FUNCTION_BLOCK FB_TouchProbe_Home_Bylimit
VAR_INPUT	
		bCMD_HomeExecute			:REFERENCE TO BOOL;			(* 执行回零*)
		bCMD_Reset					:REFERENCE TO BOOL;			(* 回零错误复位*)
		bCMD_EnableState			:BOOL;						(* 使能状态输入*)	
		bCMD_StartHomeIndex			:BOOL;						(* 是否使用索引回零*)
		eCMD_HomeDirection			:MC_Direction;				(* 回原点方向*)
		bCMD_PositiveLimit			:BOOL;						(* 正限位传感器*)
		bCMD_NegativeLimit			:BOOL;						(* 负限位传感器*)
		rCMD_HomePosition			:LREAL;						(* 设定回原点位置*)
		rCMD_TowardsVelSetValue		:LREAL;						(* 靠近原点速度*)
		rCMD_OffVelSetValue			:LREAL;						(* 离开原点速度*)
	    stHomeAdsGroup				:ST_HomeAdsGroup;			(* ADS地址信息*)

END_VAR
VAR_OUTPUT
		bResult_HomeDone			:BOOL;						(* 回原点完成状态*)
		bResult_HomeBusy			:BOOL;						(* 正在回原点中状态*)
		bResult_HomeError			:BOOL;						(* 回原点错误状态*)
		nResult_HomeErrorID			:UDINT;						(* 回原点错误代码*)
END_VAR
VAR_IN_OUT
		axis						:AXIS_REF;
END_VAR
VAR
	  
		mcHome						:MC_Home;
		mcReset						:MC_Reset;
		fbReadParameter				:ARRAY [0..4] OF ADSREAD;
		fbwriteParameter			:ARRAY [0..4] OF ADSWRITE;
		rTowardsVelActValue			:LREAL;		
		rOffVelActValue				:LREAL;
		nHomeSenorSetValue			:INT;
		nHomeSensorActValue			:INT;
		nHomeSynSetValue			:WORD;
		nHomeSynActValue			:WORD;
		nHomeSetRefMode				:DINT;
		nHomeActRefMode				:DINT;
		mcHomeStatus				:ST_McOutputs;
		fbReadParaStatus			:ARRAY [0..4] OF ST_McOutputs;
		fbWriteParaStatus			:ARRAY [0..4] OF ST_McOutputs;
		posEdge_bCMD_HomeExecute	:R_TRIG;
		posEdge_bCMD_Reset			:R_TRIG;
		negEdge_bCMD_Calibration	:F_TRIG;
		ton_bCMD_HomeExecute		:TON;
		ton_nStep					:TON;
		ton_bCMD_Reset				:TON;
		ton_McReset					:TON;
		ton_HomErr                  :TON;
		nStep						:E_HomeStep;
		mcMoveAbs					:MC_MoveAbsolute;
END_VAR

posEdge_bCMD_HomeExecute(CLK:=bCMD_HomeExecute AND bCMD_EnableState AND NOT bResult_HomeError AND NOT bResult_HomeBusy);
ton_bCMD_HomeExecute(IN:=bCMD_HomeExecute,PT:=T#100MS);

IF posEdge_bCMD_HomeExecute.Q  THEN
	nStep:=AckHomeDirection;
ELSIF	ton_bCMD_HomeExecute.Q THEN
	 bCMD_HomeExecute:=FALSE;
END_IF


IF eCMD_HomeDirection=MC_Direction.MC_Positive_Direction  THEN
	mcHome.bCalibrationCam:=bCMD_PositiveLimit;
ELSIF eCMD_HomeDirection=MC_Direction.MC_Negative_Direction THEN
		mcHome.bCalibrationCam:=bCMD_NegativeLimit;
END_IF

CASE nStep OF
IndexHomeInital:
	ton_nStep(IN:=FALSE);		
	bResult_HomeBusy:=FALSE;
	mcHome.Execute:=FALSE;
	mcMoveAbs.Execute:=FALSE;
	fbReadParameter[0].READ:=fbReadParameter[1].READ:=fbReadParameter[2].READ:=fbReadParameter[3].READ:=fbReadParameter[4].READ:=FALSE;
	fbwriteParameter[0].WRITE:=fbwriteParameter[1].WRITE:=fbwriteParameter[2].WRITE:=fbwriteParameter[3].WRITE:=fbwriteParameter[4].WRITE:=FALSE;
	IF axis.Status.Error OR mcHome.Error THEN
		nStep:=IndexHomeErrorState;
	END_IF
AckHomeDirection:
	bResult_HomeBusy:=TRUE;
	bResult_HomeDone:=FALSE;
	IF bCMD_StartHomeIndex THEN
		nHomeSetRefMode:=2;
	ELSE
		nHomeSetRefMode:=0;  
	END_IF
	IF eCMD_HomeDirection=MC_Direction.MC_Positive_Direction   THEN
		nHomeSenorSetValue:=0;
		nHomeSynSetValue:=1;
		nStep:=SetParameter;
	ELSIF eCMD_HomeDirection=MC_Direction.MC_Negative_Direction THEN
		nHomeSenorSetValue:=1;
		nHomeSynSetValue:=0;
		nStep:=SetParameter;
	ELSE
		nStep:=IndexHomeErrorState;
	END_IF
SetParameter:
	fbwriteParameter[0].WRITE:=fbwriteParameter[1].WRITE:=fbwriteParameter[2].WRITE:=
	fbwriteParameter[3].WRITE:=fbwriteParameter[4].WRITE:=TRUE;
	nStep:=SetParameterState;	
SetParameterState:
	ton_nStep(IN:=TRUE,PT:=T#100MS);
	IF ton_nStep.Q AND NOT fbWriteParaStatus[0].Busy AND NOT fbWriteParaStatus[1].Busy AND NOT fbWriteParaStatus[2].Busy AND 
		NOT fbWriteParaStatus[3].BUSY AND NOT fbWriteParaStatus[4].BUSY  THEN
		nStep:=ReadParameter;
		fbwriteParameter[0].WRITE:=fbwriteParameter[1].WRITE:=fbwriteParameter[2].WRITE
		:=fbwriteParameter[3].WRITE:=fbwriteParameter[4].WRITE:=FALSE;
	ELSIF ton_nStep.Q AND (fbWriteParaStatus[0].Error OR fbWriteParaStatus[1].Error OR fbWriteParaStatus[2].Error OR
		fbWriteParaStatus[3].Error OR fbWriteParaStatus[4].Error) THEN
		nStep:=IndexHomeErrorState;
	END_IF
ReadParameter:
	fbReadParameter[0].READ:=fbReadParameter[1].READ:=fbReadParameter[2].READ:=
	fbReadParameter[3].READ:=fbReadParameter[4].READ:=TRUE;
	nStep:=ReadParameterState;
ReadParameterState:
	ton_nStep(IN:=TRUE,PT:=T#100MS);
	
	IF ton_nStep.Q AND NOT fbReadParaStatus[0].BUSY AND NOT fbReadParaStatus[1].BUSY AND NOT fbReadParaStatus[2].BUSY
		AND NOT fbReadParaStatus[3].BUSY AND NOT fbReadParaStatus[4].BUSY THEN
		fbReadParameter[0].READ:=fbReadParameter[1].READ:=fbReadParameter[2].READ:=
		fbReadParameter[3].READ:=fbReadParameter[4].READ:=FALSE;
		nStep:=AckParameter;
	ELSIF ton_nStep.Q AND (fbReadParaStatus[0].Error OR fbReadParaStatus[1].Error OR fbReadParaStatus[2].Error OR 
		fbReadParaStatus[3].Error OR fbReadParaStatus[4].Error) THEN
		nStep:=IndexHomeErrorState;
	END_IF
AckParameter:
	IF rTowardsVelActValue=rCMD_TowardsVelSetValue AND rOffVelActValue=rCMD_OffVelSetValue AND
		nHomeSensorActValue=nHomeSenorSetValue AND nHomeSynActValue=nHomeSynSetValue 
		AND nHomeActRefMode=nHomeSetRefMode  THEN
		nStep:=ExecuteToOrigin;
	ELSE
		nStep:=IndexHomeErrorState;
	END_IF
ExecuteToOrigin:
	mcHome.Execute:=TRUE;
	nStep:=HomeMonitorState;
HomeMonitorState:
	IF mcHome.Done THEN
		mcHome.Execute:=FALSE;
		nStep:=HomeMoveABS;
	ELSIF mcHome.Error OR axis.Status.Error THEN
		nStep:=IndexHomeErrorState;
	END_IF	
	IF eCMD_HomeDirection=MC_Direction.MC_Positive_Direction AND bCMD_NegativeLimit AND ton_HomErr.Q THEN
		mcReset.Execute:=TRUE;
		nStep:=IndexHomeErrorState;
	ELSIF eCMD_HomeDirection=MC_Direction.MC_Negative_Direction AND bCMD_PositiveLimit AND ton_HomErr.Q THEN
		mcReset.Execute:=TRUE;
		nStep:=IndexHomeErrorState;
	END_IF
HomeMoveABS:
	mcMoveAbs.Execute:=TRUE;	
	IF mcMoveAbs.Done THEN
		mcMoveAbs.Execute:=FALSE;
		nStep:=ExecuteHomeDone;
	ELSIF axis.Status.Error OR mcMoveAbs.Error THEN
		nStep:=IndexHomeErrorState;
	END_IF
ExecuteHomeDone:
	bResult_HomeBusy:=FALSE;
	bResult_HomeDone:=TRUE;
	nStep:=E_HomeStep.IndexHomeInital;
IndexHomeErrorState:
	bResult_HomeBusy:=FALSE;
	bResult_HomeDone:=FALSE;
	bResult_HomeError:=TRUE;
	mcHome.Execute:=FALSE;
	mcMoveAbs.Execute:=FALSE;
	nStep:=IndexHomeInital;
END_CASE
// 超时定时器
ton_HomErr(IN:=bResult_HomeBusy , PT:=T#20S , Q=> , ET=> );

ACT_AxisControl();
ACT_ErrorID();
ACT_Reset();

ACTION ACT_AxisControl:
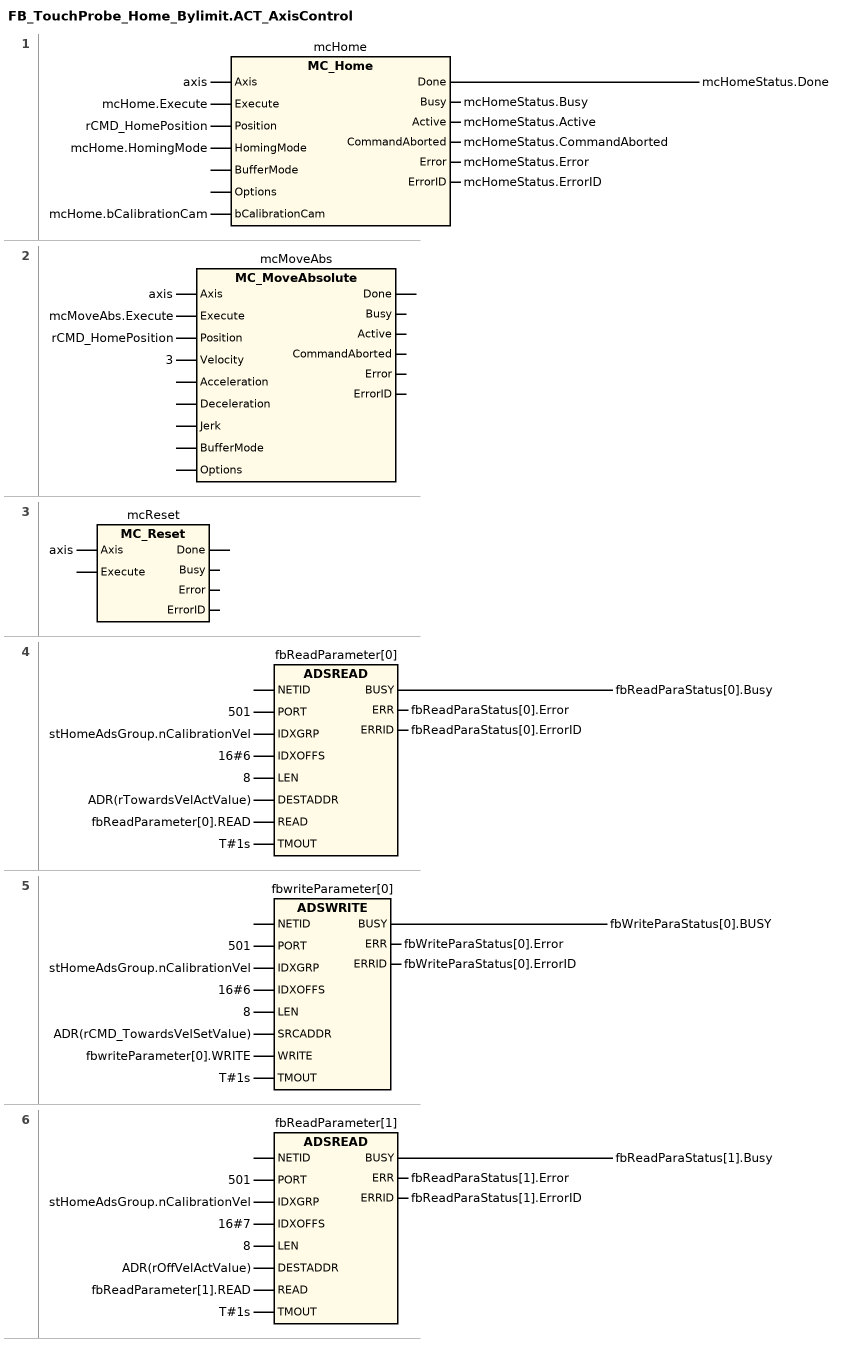
// NETWORK 1
mcHome(
    Axis := axis,
    Execute := mcHome.Execute,
    Position := rCMD_HomePosition,
    HomingMode := mcHome.HomingMode,
    bCalibrationCam := mcHome.bCalibrationCam,
    Busy => mcHomeStatus.Busy,
    Active => mcHomeStatus.Active,
    CommandAborted => mcHomeStatus.CommandAborted,
    Error => mcHomeStatus.Error,
    ErrorID => mcHomeStatus.ErrorID); // MC_Home
mcHomeStatus.Done := mcHome.Done;

// NETWORK 2
mcMoveAbs(Axis := axis, Execute := mcMoveAbs.Execute, Position := rCMD_HomePosition, Velocity := 3); // MC_MoveAbsolute

// NETWORK 3
mcReset(Axis := axis); // MC_Reset

// NETWORK 4
fbReadParameter[0](
    PORT := 501,
    IDXGRP := stHomeAdsGroup.nCalibrationVel,
    IDXOFFS := 16#6,
    LEN := 8,
    DESTADDR := ADR(rTowardsVelActValue),
    READ := fbReadParameter[0].READ,
    TMOUT := T#1s,
    ERR => fbReadParaStatus[0].Error,
    ERRID => fbReadParaStatus[0].ErrorID); // ADSREAD
fbReadParaStatus[0].Busy := fbReadParameter[0].BUSY;

// NETWORK 5
fbwriteParameter[0](
    PORT := 501,
    IDXGRP := stHomeAdsGroup.nCalibrationVel,
    IDXOFFS := 16#6,
    LEN := 8,
    SRCADDR := ADR(rCMD_TowardsVelSetValue),
    WRITE := fbwriteParameter[0].WRITE,
    TMOUT := T#1s,
    ERR => fbWriteParaStatus[0].Error,
    ERRID => fbWriteParaStatus[0].ErrorID); // ADSWRITE
fbWriteParaStatus[0].BUSY := fbwriteParameter[0].BUSY;

// NETWORK 6
fbReadParameter[1](
    PORT := 501,
    IDXGRP := stHomeAdsGroup.nCalibrationVel,
    IDXOFFS := 16#7,
    LEN := 8,
    DESTADDR := ADR(rOffVelActValue),
    READ := fbReadParameter[1].READ,
    TMOUT := T#1s,
    ERR => fbReadParaStatus[1].Error,
    ERRID => fbReadParaStatus[1].ErrorID); // ADSREAD
fbReadParaStatus[1].Busy := fbReadParameter[1].BUSY;

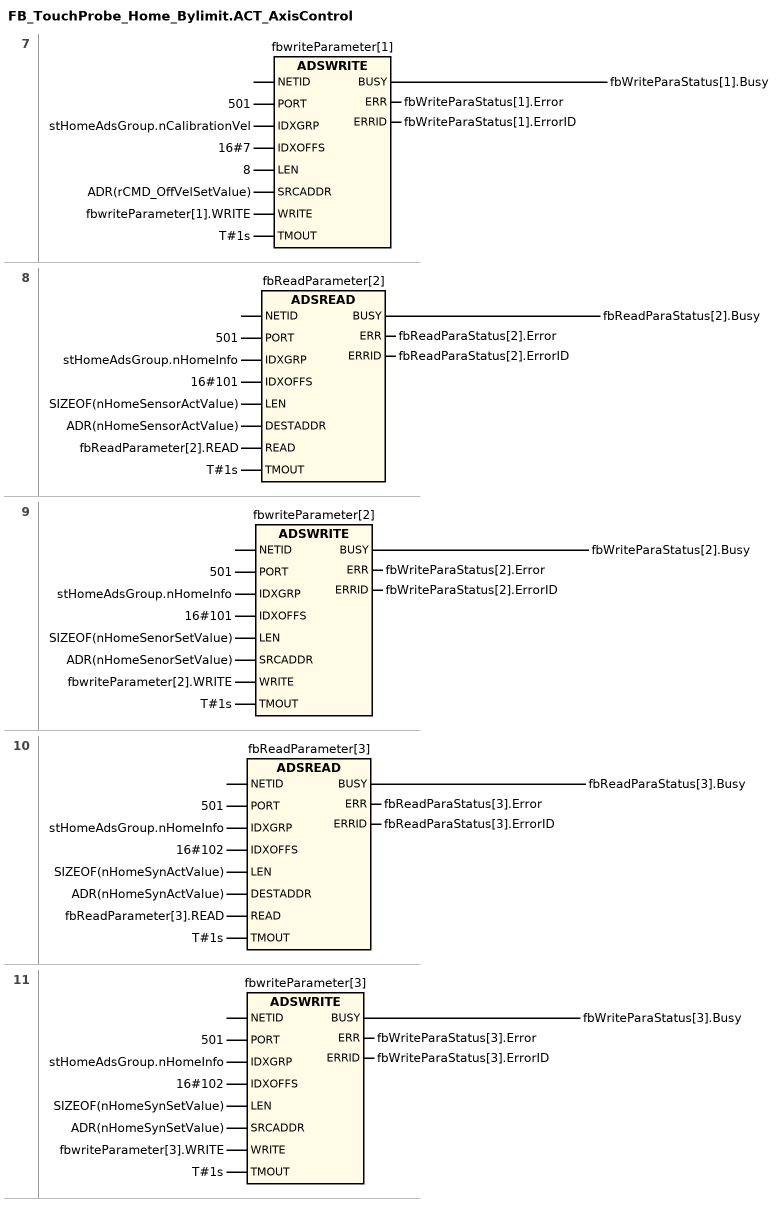
// NETWORK 7
fbwriteParameter[1](
    PORT := 501,
    IDXGRP := stHomeAdsGroup.nCalibrationVel,
    IDXOFFS := 16#7,
    LEN := 8,
    SRCADDR := ADR(rCMD_OffVelSetValue),
    WRITE := fbwriteParameter[1].WRITE,
    TMOUT := T#1s,
    ERR => fbWriteParaStatus[1].Error,
    ERRID => fbWriteParaStatus[1].ErrorID); // ADSWRITE
fbWriteParaStatus[1].Busy := fbwriteParameter[1].BUSY;

// NETWORK 8
fbReadParameter[2](
    PORT := 501,
    IDXGRP := stHomeAdsGroup.nHomeInfo,
    IDXOFFS := 16#101,
    LEN := SIZEOF(nHomeSensorActValue),
    DESTADDR := ADR(nHomeSensorActValue),
    READ := fbReadParameter[2].READ,
    TMOUT := T#1s,
    ERR => fbReadParaStatus[2].Error,
    ERRID => fbReadParaStatus[2].ErrorID); // ADSREAD
fbReadParaStatus[2].Busy := fbReadParameter[2].BUSY;

// NETWORK 9
fbwriteParameter[2](
    PORT := 501,
    IDXGRP := stHomeAdsGroup.nHomeInfo,
    IDXOFFS := 16#101,
    LEN := SIZEOF(nHomeSenorSetValue),
    SRCADDR := ADR(nHomeSenorSetValue),
    WRITE := fbwriteParameter[2].WRITE,
    TMOUT := T#1s,
    ERR => fbWriteParaStatus[2].Error,
    ERRID => fbWriteParaStatus[2].ErrorID); // ADSWRITE
fbWriteParaStatus[2].Busy := fbwriteParameter[2].BUSY;

// NETWORK 10
fbReadParameter[3](
    PORT := 501,
    IDXGRP := stHomeAdsGroup.nHomeInfo,
    IDXOFFS := 16#102,
    LEN := SIZEOF(nHomeSynActValue),
    DESTADDR := ADR(nHomeSynActValue),
    READ := fbReadParameter[3].READ,
    TMOUT := T#1s,
    ERR => fbReadParaStatus[3].Error,
    ERRID => fbReadParaStatus[3].ErrorID); // ADSREAD
fbReadParaStatus[3].Busy := fbReadParameter[3].BUSY;

// NETWORK 11
fbwriteParameter[3](
    PORT := 501,
    IDXGRP := stHomeAdsGroup.nHomeInfo,
    IDXOFFS := 16#102,
    LEN := SIZEOF(nHomeSynSetValue),
    SRCADDR := ADR(nHomeSynSetValue),
    WRITE := fbwriteParameter[3].WRITE,
    TMOUT := T#1s,
    ERR => fbWriteParaStatus[3].Error,
    ERRID => fbWriteParaStatus[3].ErrorID); // ADSWRITE
fbWriteParaStatus[3].Busy := fbwriteParameter[3].BUSY;

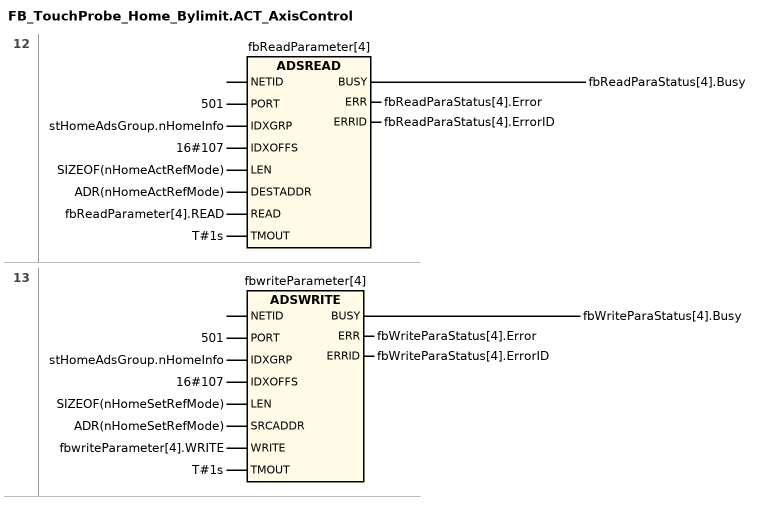
// NETWORK 12
fbReadParameter[4](
    PORT := 501,
    IDXGRP := stHomeAdsGroup.nHomeInfo,
    IDXOFFS := 16#107,
    LEN := SIZEOF(nHomeActRefMode),
    DESTADDR := ADR(nHomeActRefMode),
    READ := fbReadParameter[4].READ,
    TMOUT := T#1s,
    ERR => fbReadParaStatus[4].Error,
    ERRID => fbReadParaStatus[4].ErrorID); // ADSREAD
fbReadParaStatus[4].Busy := fbReadParameter[4].BUSY;

// NETWORK 13
fbwriteParameter[4](
    PORT := 501,
    IDXGRP := stHomeAdsGroup.nHomeInfo,
    IDXOFFS := 16#107,
    LEN := SIZEOF(nHomeSetRefMode),
    SRCADDR := ADR(nHomeSetRefMode),
    WRITE := fbwriteParameter[4].WRITE,
    TMOUT := T#1s,
    ERR => fbWriteParaStatus[4].Error,
    ERRID => fbWriteParaStatus[4].ErrorID); // ADSWRITE
fbWriteParaStatus[4].Busy := fbwriteParameter[4].BUSY;
END_ACTION

ACTION ACT_ErrorID:
nResult_HomeErrorID:=mcHome.ErrorID;
END_ACTION

ACTION ACT_Reset:
posEdge_bCMD_Reset(CLK:=bCMD_Reset);
ton_bCMD_Reset(IN:=bCMD_Reset,PT:=T#100MS);
ton_McReset(IN:=mcReset.Execute,PT:=T#100MS);
IF posEdge_bCMD_Reset.Q THEN
	bResult_HomeBusy:=FALSE;
	bResult_HomeDone:=FALSE;
	bResult_HomeError:=FALSE;
	nStep:=IndexHomeInital;
	mcReset.Execute:=TRUE;
	mcMoveAbs.Execute:=FALSE;
ELSIF ton_bCMD_Reset.Q THEN
	bCMD_Reset:=FALSE;
END_IF

IF ton_McReset.Q THEN
	mcReset.Execute:=FALSE;
END_IF
END_ACTION

END_FUNCTION_BLOCK

(* stored: Version 1.1.0.1, ProductVersion 3.1.4024.12
   POU FB_TouchProbe_Home_Bylimit: Id {2ef58b1e-4663-40e7-8041-e93620483a0f}, SpecialFunc None
   Action ACT_AxisControl: Id {7f291c64-624f-4e3c-b7dc-940e1cd2bb23}
   Action ACT_ErrorID: Id {b9945f03-c3b3-42eb-8097-b00eaa196762}
   Action ACT_Reset: Id {85e9d134-bfb8-4697-bb14-48a7732438f9} *)
